// TIA Portal project "Kacper_Siemianowski_ALGORITHMIC" (V16)

(* hardware
DEVICE "S71500/ET200MP station_1"  S7-1500 station
   slot 0: "Rail_0"  Rack  6ES7 590-1***0-0AA0
   slot 1: "6GK7 513-1AL00-0AB0"  CPU 1513-1 PN  6ES7 513-1AL00-0AB0  V1.8
      slot 3: "CPU display_1"  6ES7591-1AA00-0AA0
      slot 32768: "PROFINET interface_1"  X1
         slot 32769: "Port_1"  X1 P1
         slot 32770: "Port_2"  X1 P2
   slot 2: "DI 16x24VDC / DQ 16x24VDC/0.5A BA_1"  DI 16x24VDC/DQ 16x24VDC/0.5A BA  6ES7 523-1BL00-0AA0  V1.1
   slot 3: "AI 4xU/I/RTD/TC / AQ 2xU/I ST_1"  AI/AQ 4xU/I/RTD/TC / 2xU/I ST  6ES7 534-7QE00-0AB0  V1.0
*)

// ===== PLC "6GK7 513-1AL00-0AB0"  CPU 1513-1 PN =====

VAR_GLOBAL   // PLC tag table "main"
   "Przycisk monostabilny - Button1" AT %I0.0 : Bool;   // przycisk piesi 1
   "Przycisk monostabilny - Button2" AT %I0.1 : Bool;   // przycisk piesi 2
   "Pomiar prędkości SpeedCamera1: 0-200 [km/h]" AT %IW2 : Int;
   "Pomiar natężenia ruchu: 0-100 [pojazdów/min]" AT %IW4 : Int;
   "Światło czerwone sygnalizacji świetlnej - TrafficLight1" AT %Q0.0 : Bool;
   "Światło żółte sygnalizacji świetlnej - TrafficLight1" AT %Q0.1 : Bool;
   "Światło zielone sygnalizacji świetlnej - TrafficLight1" AT %Q0.2 : Bool;
   "Sygnalizacja dźwiękowa świateł dla pieszych - Buzzer1" AT %Q0.3 : Bool;
   "Sygnalizacja dźwiękowa świateł dla pieszych - Buzzer2" AT %Q0.4 : Bool;
   "Światło zielone sygnalizacji świetlnej dla pieszych - PedestrianLight1" AT %Q0.5 : Bool;
   "Światło czerwone sygnalizacji świetlnej dla pieszych - PedestrianLight1" AT %Q0.6 : Bool;
   "Światło zielone sygnalizacji świetlnej dla pieszych - PedestrianLight2" AT %Q0.7 : Bool;
   "Światło czerwone sygnalizacji świetlnej dla pieszych - PedestrianLight2" AT %Q1.0 : Bool;
   "Tag_1" AT %M20.0 : Bool;
   "Clock_Byte" AT %MB0 : Byte;
   "Clock_10Hz" AT %M0.0 : Bool;
   "Clock_5Hz" AT %M0.1 : Bool;
   "Clock_2.5Hz" AT %M0.2 : Bool;
   "Clock_2Hz" AT %M0.3 : Bool;
   "Clock_1.25Hz" AT %M0.4 : Bool;
   "Clock_1Hz" AT %M0.5 : Bool;
   "Clock_0.625Hz" AT %M0.6 : Bool;
   "Clock_0.5Hz" AT %M0.7 : Bool;
END_VAR

VAR_GLOBAL   // PLC tag table "test"
   "Przycisk monostabilny - Button1(test)" AT %M10.0 : Bool;   // przycisk piesi 1
   "Przycisk monostabilny - Button2(test)" AT %M10.1 : Bool;   // przycisk piesi 2
   "Pomiar prędkości SpeedCamera1: 0-200 [km/h](test)" AT %MW12 : Int;
   "Pomiar natężenia ruchu: 0-100 [pojazdów/min](test)" AT %MW14 : Int;
END_VAR

DATA_BLOCK "Kacper_Siemianowski_ALGORITHMIC_FB_DB"   // DB1
{ S7_Optimized_Access := 'TRUE' }
VERSION : 0.1
// stored: InstanceOfName Kacper_Siemianowski_ALGORITHMIC_FB
"Kacper_Siemianowski_ALGORITHMIC_FB"
BEGIN
END_DATA_BLOCK

// folder: System blocks/Program resources

DATA_BLOCK "IEC_Timer_0_DB"   // DB2
{ S7_Optimized_Access := 'TRUE' }
AUTHOR : Simatic
FAMILY : IEC
NAME : IEC_TMR
VERSION : 1.0
// stored: InstanceOfName IEC_TIMER
"IEC_TIMER"
BEGIN
END_DATA_BLOCK

DATA_BLOCK "IEC_Timer_0_DB_1"   // DB3
{ S7_Optimized_Access := 'TRUE' }
AUTHOR : Simatic
FAMILY : IEC
NAME : IEC_TMR
VERSION : 1.0
// stored: InstanceOfName IEC_TIMER
"IEC_TIMER"
BEGIN
END_DATA_BLOCK

DATA_BLOCK "IEC_Timer_0_DB_2"   // DB4
{ S7_Optimized_Access := 'TRUE' }
AUTHOR : Simatic
FAMILY : IEC
NAME : IEC_TMR
VERSION : 1.0
// stored: InstanceOfName IEC_TIMER
"IEC_TIMER"
BEGIN
END_DATA_BLOCK

DATA_BLOCK "IEC_Timer_0_DB_3"   // DB5
{ S7_Optimized_Access := 'TRUE' }
AUTHOR : Simatic
FAMILY : IEC
NAME : IEC_TMR
VERSION : 1.0
// stored: InstanceOfName IEC_TIMER
"IEC_TIMER"
BEGIN
END_DATA_BLOCK

DATA_BLOCK "IEC_Timer_0_DB_4"   // DB6
{ S7_Optimized_Access := 'TRUE' }
AUTHOR : Simatic
FAMILY : IEC
NAME : IEC_TMR
VERSION : 1.0
// stored: InstanceOfName IEC_TIMER
"IEC_TIMER"
BEGIN
END_DATA_BLOCK

DATA_BLOCK "IEC_Timer_0_DB_6"   // DB8
{ S7_Optimized_Access := 'TRUE' }
AUTHOR : Simatic
FAMILY : IEC
NAME : IEC_TMR
VERSION : 1.0
// stored: InstanceOfName IEC_TIMER
"IEC_TIMER"
BEGIN
END_DATA_BLOCK

// folder: (top level)

FUNCTION_BLOCK "Kacper_Siemianowski_ALGORITHMIC_FB"   // FB1, LAD
{ S7_Optimized_Access := 'TRUE' }
VERSION : 0.1
   VAR_INPUT
      pedestrianButton1 : Bool;   // Przycisk monostabilny - Button1
      pedestrianButton2 : Bool;   // Przycisk monostabilny - Button2
      speedValue1 : Int;   // Pomiar prędkości SpeedCamera1: 0-200 [km/h]
      TrafficIntensity1 : Int;   // Pomiar natężenia ruchu: 0-100 [pojazdów/min]
   END_VAR
   VAR_OUTPUT
      redTrafficLight1 : Bool;   // Światło czerwone sygnalizacji świetlnej - TrafficLight1
      yellowTrafficLight1 : Bool;   // Światło żółte sygnalizacji świetlnej - TrafficLight1
      greenTrafficLight1 : Bool;   // Światło zielone sygnalizacji świetlnej - TrafficLight1
      buzzer1 : Bool;   // Sygnalizacja dźwiękowa świateł dla pieszych - Buzzer1
      buzzer2 : Bool;   // Sygnalizacja dźwiękowa świateł dla pieszych - Buzzer2
      redPedestrianLight1 : Bool;   // Światło czerwone sygnalizacji świetlnej dla pieszych - PedestrianLight1
      greenPedestrianLight1 : Bool;   // Światło zielone sygnalizacji świetlnej dla pieszych - PedestrianLight1
      redPedestrianLight2 : Bool;   // Światło czerwone sygnalizacji świetlnej dla pieszych - PedestrianLight2
      greenPedestrianLight2 : Bool;   // Światło zielone sygnalizacji świetlnej dla pieszych - PedestrianLight2
   END_VAR
   VAR
      ActualSpeed : Int;
      ActualIntensity : Int;
      SpeedLimit : Int := 50;
      Temp_1 : Real;
      Temp_2 : Real;
      OverLimitedSpeed : Bool;
      ButtonActivated : Bool;
      WaitingTime : Time;   // [s]
      Temp_3 : Int;
      WaitingTimePassed : Bool;
      TraficStop : Bool;
      Temp_4 : Bool;
      YellowLight1 : Bool;
      RedLight1 : Bool;
      Temp_5 : Bool;
      Temp_6 : Bool;
      Temp_7 : Bool;
      GreenPedestrianM : Bool;
      GreenPedestrianBlinking : Bool;
      Temp_8 : Bool;
      RedPedestrianM : Bool;
      YellowLight2 : Bool;
      Temp_9 : Bool;
      GreenLight1 : Bool;
      Temp_10 : Bool;
      Temp_11 : Bool;
      Temp_12 : Bool;
      Temp_13 : Bool;
      Temp_14 : Bool;
      Temp_15 : Bool;
      Temp_16 : Bool;
      Temp_17 : Bool;
   END_VAR
   VAR_TEMP   // added for the SCL form of the ladder/FBD networks
      _w1 : Bool;
   END_VAR
BEGIN

REGION Network 1: Skalowanie prędkości
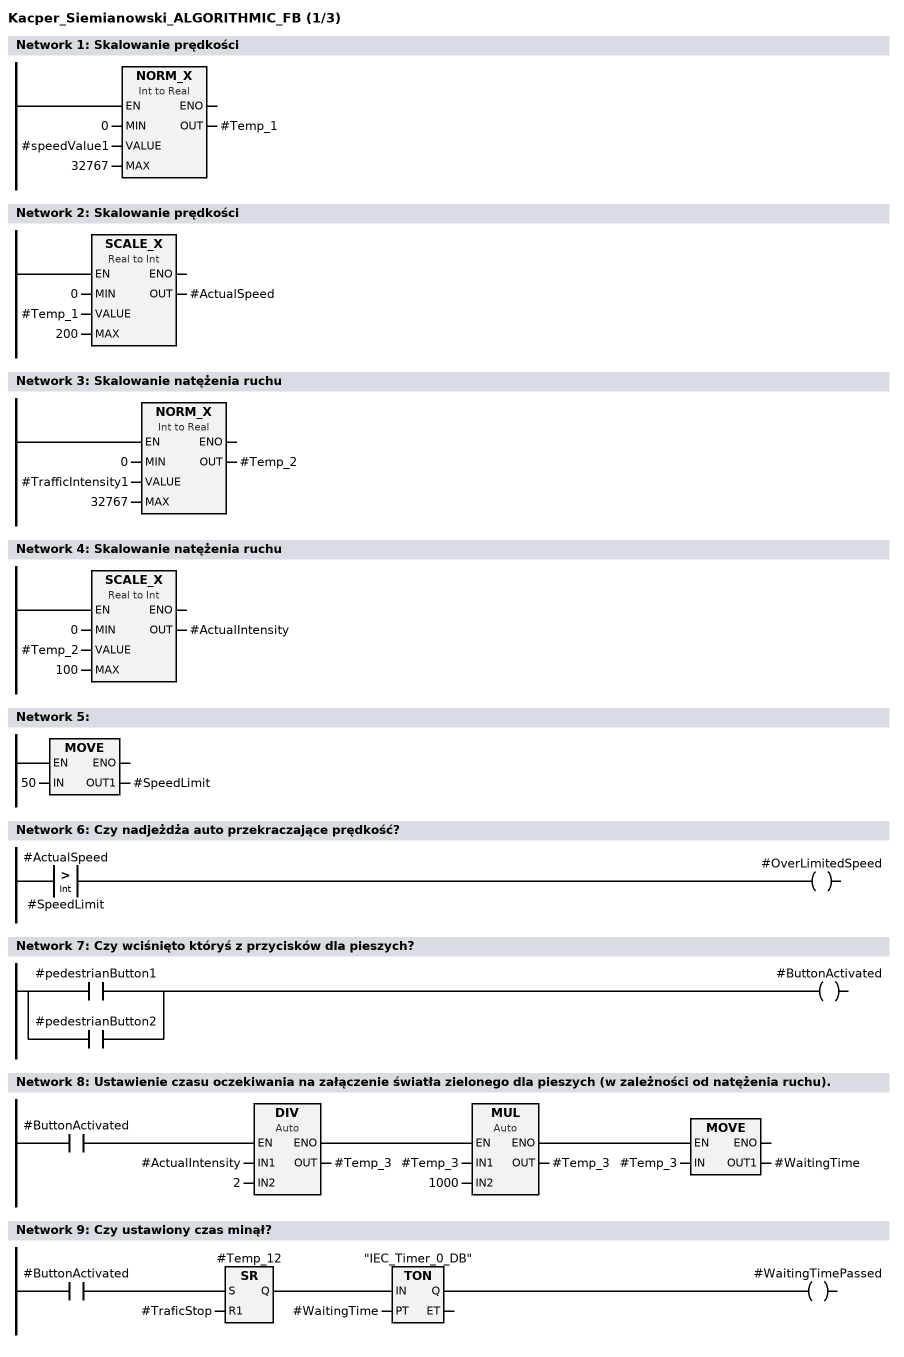
   RUNG wire#powerrail
      { S7_Templates := "[SrcType := Int, DestType := Real]" } Normalize(min := 0, value := #speedValue1, max := 32767, out => #Temp_1)
   END_RUNG
   // the same network as SCL:
   #Temp_1 := NORM_X(MIN := 0, VALUE := #speedValue1, MAX := 32767);
END_REGION

REGION Network 2: Skalowanie prędkości
   RUNG wire#powerrail
      { S7_Templates := "[SrcType := Real, DestType := Int]" } Scale(min := 0, value := #Temp_1, max := 200, out => #ActualSpeed)
   END_RUNG
   // the same network as SCL:
   #ActualSpeed := SCALE_X(MIN := 0, VALUE := #Temp_1, MAX := 200);
END_REGION

REGION Network 3: Skalowanie natężenia ruchu
   RUNG wire#powerrail
      { S7_Templates := "[SrcType := Int, DestType := Real]" } Normalize(min := 0, value := #TrafficIntensity1, max := 32767, out => #Temp_2)
   END_RUNG
   // the same network as SCL:
   #Temp_2 := NORM_X(MIN := 0, VALUE := #TrafficIntensity1, MAX := 32767);
END_REGION

REGION Network 4: Skalowanie natężenia ruchu
   RUNG wire#powerrail
      { S7_Templates := "[SrcType := Real, DestType := Int]" } Scale(min := 0, value := #Temp_2, max := 100, out => #ActualIntensity)
   END_RUNG
   // the same network as SCL:
   #ActualIntensity := SCALE_X(MIN := 0, VALUE := #Temp_2, MAX := 100);
END_REGION

REGION Network 5
   RUNG wire#powerrail
      Move(in := 50, out1 => #SpeedLimit)
   END_RUNG
   // the same network as SCL:
   #SpeedLimit := 50;
END_REGION

REGION Network 6: Czy nadjeżdża auto przekraczające prędkość?
   RUNG wire#powerrail
      { S7_Templates := "SrcType := Int" } GT_Contact(in1 := #ActualSpeed, in2 := #SpeedLimit)
      Coil( #OverLimitedSpeed )
   END_RUNG
   // the same network as SCL:
   #OverLimitedSpeed := #ActualSpeed > #SpeedLimit;
END_REGION

REGION Network 7: Czy wciśnięto któryś z przycisków dla pieszych?
   RUNG wire#powerrail
      Contact( #pedestrianButton1 )
      wire#w1
      Coil( #ButtonActivated )
   END_RUNG
   RUNG wire#powerrail
      Contact( #pedestrianButton2 )
   END_RUNG wire#w1
   // the same network as SCL:
   #ButtonActivated := #pedestrianButton1 OR #pedestrianButton2;
END_REGION

REGION Network 8: Ustawienie czasu oczekiwania na załączenie światła zielonego dla pieszych (w zależności od natężenia ruchu).
   RUNG wire#powerrail
      Contact( #ButtonActivated )
      Div(in1 := #ActualIntensity, in2 := 2, out => #Temp_3)
      Mul(in1 := #Temp_3, in2 := 1000, out => #Temp_3)
      Move(in := #Temp_3, out1 => #WaitingTime)
   END_RUNG
   // the same network as SCL:
   IF #ButtonActivated THEN
       #Temp_3 := #ActualIntensity / 2;
       #Temp_3 := #Temp_3 * 1000;
       #WaitingTime := #Temp_3;
   END_IF;
END_REGION

REGION Network 9: Czy ustawiony czas minął?
   IF #ButtonActivated THEN
       #Temp_12 := TRUE;   // SR flip-flop
   END_IF;
   IF #TraficStop THEN #Temp_12 := FALSE; END_IF;
   "IEC_Timer_0_DB".TON(IN := #Temp_12, PT := #WaitingTime);
   #WaitingTimePassed := "IEC_Timer_0_DB".Q;
END_REGION

REGION Network 10: Zatrzymanie ruchu aut
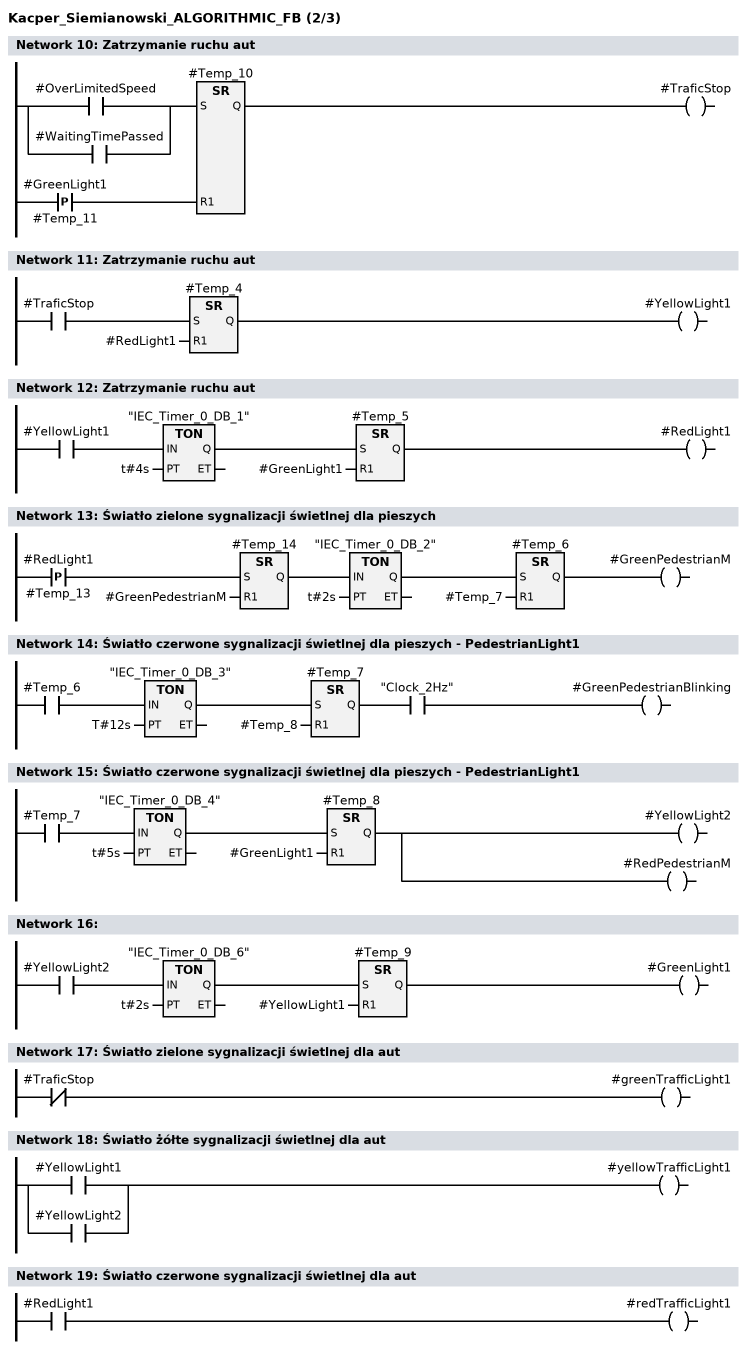
   RUNG wire#powerrail
      Contact( #OverLimitedSpeed )
      wire#w1
      S_SR(operand := #Temp_10, r1 := wire#w2)
      Coil( #TraficStop )
   END_RUNG
   RUNG wire#powerrail
      Contact( #WaitingTimePassed )
   END_RUNG wire#w1
   RUNG wire#powerrail
      P_Contact(operand := #GreenLight1, bit := #Temp_11)
   END_RUNG wire#w2
   // the same network as SCL:
   #_w1 := #GreenLight1 AND NOT #Temp_11;   // rising edge of #GreenLight1
   #Temp_11 := #GreenLight1;
   IF #OverLimitedSpeed OR #WaitingTimePassed THEN
       #Temp_10 := TRUE;   // SR flip-flop
   END_IF;
   IF #_w1 THEN #Temp_10 := FALSE; END_IF;
   #TraficStop := #Temp_10;
END_REGION

REGION Network 11: Zatrzymanie ruchu aut
   RUNG wire#powerrail
      Contact( #TraficStop )
      S_SR(operand := #Temp_4, r1 := #RedLight1)
      Coil( #YellowLight1 )
   END_RUNG
   // the same network as SCL:
   IF #TraficStop THEN
       #Temp_4 := TRUE;   // SR flip-flop
   END_IF;
   IF #RedLight1 THEN #Temp_4 := FALSE; END_IF;
   #YellowLight1 := #Temp_4;
END_REGION

REGION Network 12: Zatrzymanie ruchu aut
   "IEC_Timer_0_DB_1".TON(IN := #YellowLight1, PT := t#4s);
   IF "IEC_Timer_0_DB_1".Q THEN
       #Temp_5 := TRUE;   // SR flip-flop
   END_IF;
   IF #GreenLight1 THEN #Temp_5 := FALSE; END_IF;
   #RedLight1 := #Temp_5;
END_REGION

REGION Network 13: Światło zielone sygnalizacji świetlnej dla pieszych
   #_w1 := #RedLight1 AND NOT #Temp_13;   // rising edge of #RedLight1
   #Temp_13 := #RedLight1;
   IF #_w1 THEN
       #Temp_14 := TRUE;   // SR flip-flop
   END_IF;
   IF #GreenPedestrianM THEN #Temp_14 := FALSE; END_IF;
   "IEC_Timer_0_DB_2".TON(IN := #Temp_14, PT := t#2s);
   IF "IEC_Timer_0_DB_2".Q THEN
       #Temp_6 := TRUE;   // SR flip-flop
   END_IF;
   IF #Temp_7 THEN #Temp_6 := FALSE; END_IF;
   #GreenPedestrianM := #Temp_6;
END_REGION

REGION Network 14: Światło czerwone sygnalizacji świetlnej dla pieszych - PedestrianLight1
   "IEC_Timer_0_DB_3".TON(IN := #Temp_6, PT := T#12s);
   IF "IEC_Timer_0_DB_3".Q THEN
       #Temp_7 := TRUE;   // SR flip-flop
   END_IF;
   IF #Temp_8 THEN #Temp_7 := FALSE; END_IF;
   #GreenPedestrianBlinking := #Temp_7 AND "Clock_2Hz";
END_REGION

REGION Network 15: Światło czerwone sygnalizacji świetlnej dla pieszych - PedestrianLight1
   "IEC_Timer_0_DB_4".TON(IN := #Temp_7, PT := t#5s);
   IF "IEC_Timer_0_DB_4".Q THEN
       #Temp_8 := TRUE;   // SR flip-flop
   END_IF;
   IF #GreenLight1 THEN #Temp_8 := FALSE; END_IF;
   #YellowLight2 := #Temp_8;
   #RedPedestrianM := #Temp_8;
END_REGION

REGION Network 16
   "IEC_Timer_0_DB_6".TON(IN := #YellowLight2, PT := t#2s);
   IF "IEC_Timer_0_DB_6".Q THEN
       #Temp_9 := TRUE;   // SR flip-flop
   END_IF;
   IF #YellowLight1 THEN #Temp_9 := FALSE; END_IF;
   #GreenLight1 := #Temp_9;
END_REGION

REGION Network 17: Światło zielone sygnalizacji świetlnej dla aut
   RUNG wire#powerrail
      I_Contact( #TraficStop )
      Coil( #greenTrafficLight1 )
   END_RUNG
   // the same network as SCL:
   #greenTrafficLight1 := NOT #TraficStop;
END_REGION

REGION Network 18: Światło żółte sygnalizacji świetlnej dla aut
   RUNG wire#powerrail
      Contact( #YellowLight1 )
      wire#w1
      Coil( #yellowTrafficLight1 )
   END_RUNG
   RUNG wire#powerrail
      Contact( #YellowLight2 )
   END_RUNG wire#w1
   // the same network as SCL:
   #yellowTrafficLight1 := #YellowLight1 OR #YellowLight2;
END_REGION

REGION Network 19: Światło czerwone sygnalizacji świetlnej dla aut
   RUNG wire#powerrail
      Contact( #RedLight1 )
      Coil( #redTrafficLight1 )
   END_RUNG
   // the same network as SCL:
   #redTrafficLight1 := #RedLight1;
END_REGION

REGION Network 20: Światło zielone sygnalizacji świetlnej dla pieszych
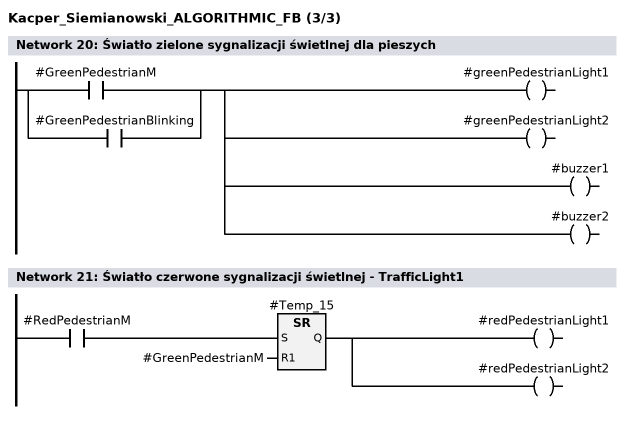
   RUNG wire#powerrail
      Contact( #GreenPedestrianM )
      wire#w1
      Coil( #greenPedestrianLight1 )
   END_RUNG
   RUNG wire#powerrail
      Contact( #GreenPedestrianBlinking )
   END_RUNG wire#w1
   RUNG wire#w1
      Coil( #greenPedestrianLight2 )
   END_RUNG
   RUNG wire#w1
      Coil( #buzzer1 )
   END_RUNG
   RUNG wire#w1
      Coil( #buzzer2 )
   END_RUNG
   // the same network as SCL:
   #greenPedestrianLight1 := #GreenPedestrianM OR #GreenPedestrianBlinking;
   #greenPedestrianLight2 := #greenPedestrianLight1;
   #buzzer1 := #greenPedestrianLight1;
   #buzzer2 := #greenPedestrianLight1;
END_REGION

REGION Network 21: Światło czerwone sygnalizacji świetlnej - TrafficLight1
   RUNG wire#powerrail
      Contact( #RedPedestrianM )
      S_SR(operand := #Temp_15, r1 := #GreenPedestrianM)
      wire#w1
      Coil( #redPedestrianLight1 )
   END_RUNG
   RUNG wire#w1
      Coil( #redPedestrianLight2 )
   END_RUNG
   // the same network as SCL:
   IF #RedPedestrianM THEN
       #Temp_15 := TRUE;   // SR flip-flop
   END_IF;
   IF #GreenPedestrianM THEN #Temp_15 := FALSE; END_IF;
   #redPedestrianLight1 := #Temp_15;
   #redPedestrianLight2 := #Temp_15;
END_REGION
END_FUNCTION_BLOCK

ORGANIZATION_BLOCK "Main"   // OB1, LAD, ProgramCycle
TITLE = "Main Program Sweep (Cycle)"
{ S7_Optimized_Access := 'TRUE' }
VERSION : 0.1
   VAR_INPUT
      Initial_Call : Bool;   // Initial call of this OB
      Remanence : Bool;   // =True, if remanent data are available
   END_VAR
BEGIN

REGION Network 1
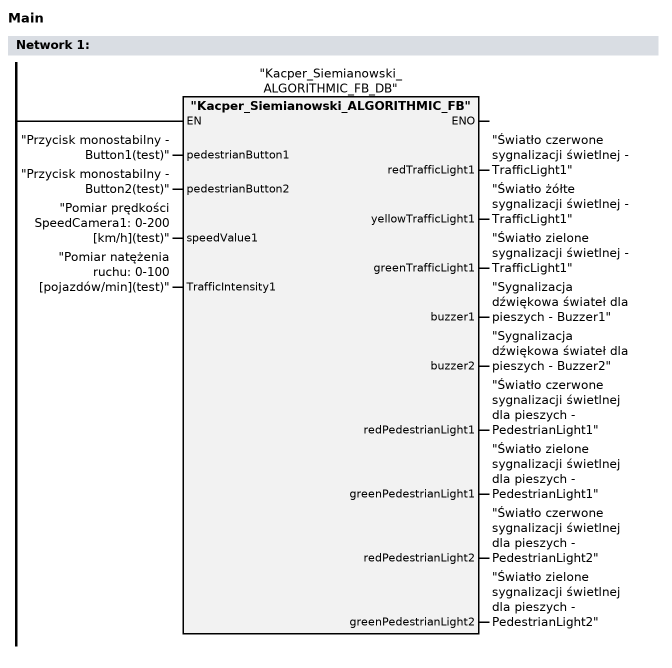
   RUNG wire#powerrail
      "Kacper_Siemianowski_ALGORITHMIC_FB_DB"(pedestrianButton1 := "Przycisk monostabilny - Button1(test)", pedestrianButton2 := "Przycisk monostabilny - Button2(test)", speedValue1 := "Pomiar prędkości SpeedCamera1: 0-200 [km/h](test)", TrafficIntensity1 := "Pomiar natężenia ruchu: 0-100 [pojazdów/min](test)", redTrafficLight1 => "Światło czerwone sygnalizacji świetlnej - TrafficLight1", yellowTrafficLight1 => "Światło żółte sygnalizacji świetlnej - TrafficLight1", greenTrafficLight1 => "Światło zielone sygnalizacji świetlnej - TrafficLight1", buzzer1 => "Sygnalizacja dźwiękowa świateł dla pieszych - Buzzer1", buzzer2 => "Sygnalizacja dźwiękowa świateł dla pieszych - Buzzer2", redPedestrianLight1 => "Światło czerwone sygnalizacji świetlnej dla pieszych - PedestrianLight1", greenPedestrianLight1 => "Światło zielone sygnalizacji świetlnej dla pieszych - PedestrianLight1", redPedestrianLight2 => "Światło czerwone sygnalizacji świetlnej dla pieszych - PedestrianLight2", greenPedestrianLight2 => "Światło zielone sygnalizacji świetlnej dla pieszych - PedestrianLight2")
   END_RUNG
   // the same network as SCL:
   "Kacper_Siemianowski_ALGORITHMIC_FB_DB"(pedestrianButton1 := "Przycisk monostabilny - Button1(test)",   // "Kacper_Siemianowski_ALGORITHMIC_FB"
                           pedestrianButton2 := "Przycisk monostabilny - Button2(test)",
                           speedValue1 := "Pomiar prędkości SpeedCamera1: 0-200 [km/h](test)",
                           TrafficIntensity1 := "Pomiar natężenia ruchu: 0-100 [pojazdów/min](test)",
                           redTrafficLight1 => "Światło czerwone sygnalizacji świetlnej - TrafficLight1",
                           yellowTrafficLight1 => "Światło żółte sygnalizacji świetlnej - TrafficLight1",
                           greenTrafficLight1 => "Światło zielone sygnalizacji świetlnej - TrafficLight1",
                           buzzer1 => "Sygnalizacja dźwiękowa świateł dla pieszych - Buzzer1",
                           buzzer2 => "Sygnalizacja dźwiękowa świateł dla pieszych - Buzzer2",
                           redPedestrianLight1 => "Światło czerwone sygnalizacji świetlnej dla pieszych - PedestrianLight1",
                           greenPedestrianLight1 => "Światło zielone sygnalizacji świetlnej dla pieszych - PedestrianLight1",
                           redPedestrianLight2 => "Światło czerwone sygnalizacji świetlnej dla pieszych - PedestrianLight2",
                           greenPedestrianLight2 => "Światło zielone sygnalizacji świetlnej dla pieszych - PedestrianLight2");
END_REGION
END_ORGANIZATION_BLOCK